FUNCTION TIME_TO_100NS : ULINT
VAR_INPUT
    nTime : TIME;
END_VAR
VAR
END_VAR

TIME_TO_100NS := TIME_TO_ULINT(nTime)*10000;

END_FUNCTION

(* stored: Version 1.1.0.1, ProductVersion 3.1.4022.18
   POU TIME_TO_100NS: Id {ee77a1b2-f30d-4a79-9ca8-80e9b00aec3d}, SpecialFunc None *)
